FUNCTION F_ComputeSInt64Size : UDINT
VAR_INPUT
    nValue  : LINT;
END_VAR


F_ComputeSInt64Size := F_ComputeRawVarint64Size(F_EncodeZigZag64(nValue));

END_FUNCTION

(* stored: Version 1.1.0.1
   POU F_ComputeSInt64Size: Id {abf6d1d4-f1e7-40d8-a715-d04005b02aea}, SpecialFunc None *)
